RoboDK station: RBT23CS013(Yashashri_Kalekar).rdk

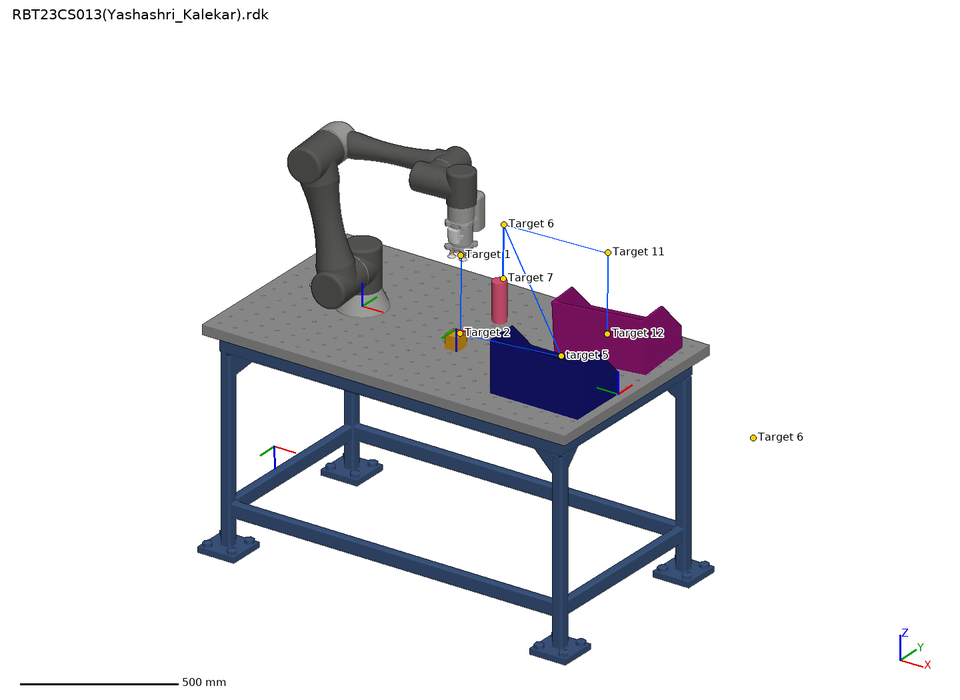
[picture v0: the station drawn from its stored meshes, robots at their saved joint values, targets as dots, program paths as lines]
Station RBT23CS013(Yashashri_Kalekar) (saved by RoboDK 5.9.2). Poses are relative to the parent item; angles as X-Y-Z fixed-axis rotations.
  - frame TM5-900 Base at (-216.63, 0, 0) mm
    - robot TM5-900: 6 axes, payload 4 kg, reach 900 mm, repeatability 0.1 mm, weight 30 kg
        modified DH rows (alpha deg, a mm, theta deg, d mm): 0, 0, 0, 145.2; 90, 0, 90, 0; 0, 429, 0, 0; 0, 411, -90, 122.3; -90, 0, 0, 106.5; 90, 0, 180, 114.15
        joint limits [-360, -180, -155, -180, -180, -270] to [360, 180, 155, 180, 180, 270]; home [0, 0, 90, -90, 90, 0]; saved at [4.776, -11.318, 99.736, 1.887, 89.639, -89.005]
      - tool SMC ZXP7A01-ZP25C-X1 Vacuum Gripper, TCP at (0, 0, 125) mm, size 88 x 106.8 x 127.9 mm
    - object Table 1400x800x800mm at (0, 0, 0) mm, size 1420 x 820 x 800 mm, geometry from Table.sld
  - frame Frame 2 at (811.01, -58.35, 0.44) mm, rotated rx 0 ry 0 rz 90.19 deg
    - object Bin Blue at (0, 0, 0) mm, size 225 x 337.5 x 191.2 mm, geometry from Bin-Blue.sld
  - frame Frame 3 at (181.66, -53.2, 51.85) mm, rotated rx -179.22 ry 0 rz 0 deg
    - object Cube 50mm at (-10, 0, 0) mm, size 50 x 50 x 50 mm, geometry from Cube.sld
    - target Target 1 (Cartesian target) at (42.39, 30.35, -286.08) mm, rotated rx 1.14 ry 0.35 rz 176.22 deg; joints [4.776, -11.318, 99.736, 1.887, 89.639, -89.005] of TM5-900
    - target Target 2 (Cartesian target) at (41.08, 35.92, -10.91) mm, rotated rx 1.14 ry 0.35 rz 176.22 deg; joints [4.546, 2.331, 129.082, -41.11, 89.638, -89.234] of TM5-900
    - target target 5 (Cartesian target) at (415.52, 10.86, -25.67) mm, rotated rx 1.14 ry 0.35 rz 176.22 deg; joints [4.198, 46.277, 61.378, -17.353, 89.636, -89.582] of TM5-900
    - object Bin Pink at (617.32, -365.19, 43.61) mm, rotated rx 177.31 ry 0 rz -94.05 deg, size 225 x 337.5 x 191.2 mm, geometry from Bin-Pink.sld
      - target Target 6 (Cartesian target) at (25.1, -231.08, -280.88) mm, rotated rx 1.14 ry 0.35 rz 176.22 deg; joints [37.917, -10.007, 98.873, 1.586, 89.865, -55.864] of TM5-900
      - target Target 6 (Cartesian target) at (25.1, -231.08, -280.88) mm, rotated rx 1.14 ry 0.35 rz 176.22 deg; joints [37.917, -10.007, 98.873, 1.586, 89.865, -55.864] of TM5-900
    - target Target 6 (Cartesian target) at (25.1, -231.08, -280.88) mm, rotated rx 1.14 ry 0.35 rz 176.22 deg; joints [37.917, -10.007, 98.873, 1.586, 89.865, -55.864] of TM5-900
    - target Target 7 (Cartesian target) at (24.19, -227.22, -89.78) mm, rotated rx 1.14 ry 0.35 rz 176.22 deg; joints [37.858, -4.045, 121.336, -26.84, 89.864, -55.923] of TM5-900
    - target Target 10 (Cartesian target) at (25.1, -231.08, -280.88) mm, rotated rx 1.14 ry 0.35 rz 176.22 deg; joints [37.917, -10.007, 98.873, 1.586, 89.865, -55.864] of TM5-900
    - target Target 11 (Cartesian target) at (408.79, -256.41, -278.53) mm, rotated rx 1.14 ry 0.35 rz 176.22 deg; joints [22.411, 53.381, 11.786, 25.233, 89.749, -71.369] of TM5-900
    - target Target 12 (Cartesian target) at (407.43, -250.65, 6.05) mm, rotated rx 1.14 ry 0.35 rz 176.22 deg; joints [22.324, 49.649, 59.362, -18.612, 89.748, -71.456] of TM5-900
    - frame Frame 4 at (0, 1000, 0) mm
      - object Cylinder 50x150mm at (18.29, -1213.2, -88.15) mm, size 50 x 50 x 150 mm, geometry from Cylinder-50x150mm.sld
  - program Prog1 (10 instructions, listed below)
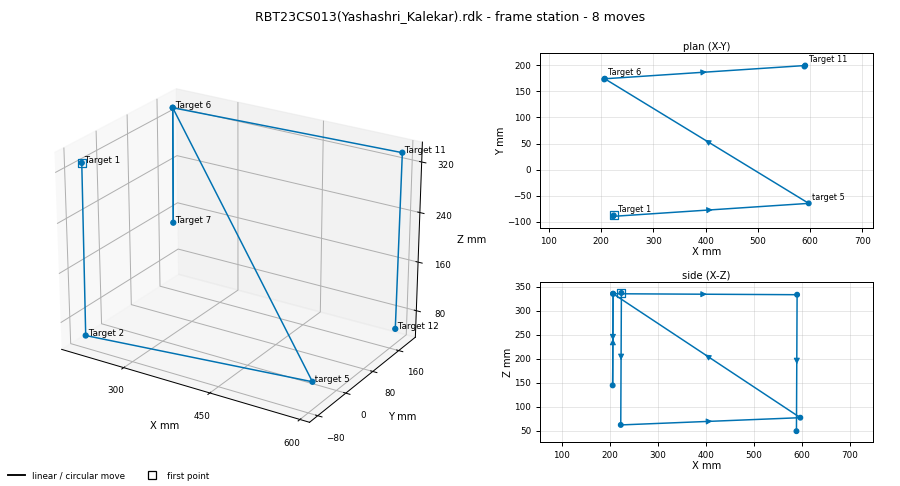
[picture p0: tool path of RBT23CS013(Yashashri_Kalekar).rdk in frame station, 8 of 8 moves have a stored position in this frame; points joined in program order, loops and branches not executed]

--- program Prog1 (robot TM5-900) ---
  Set Ref.: Frame 3
  Set Tool: SMC ZXP7A01-ZP25C-X1 Vacuum Gripper
  MoveJ (Target 1)
  MoveL (Target 2)
  MoveL (target 5)
  MoveL (Target 6)
  MoveL (Target 7)
  MoveL (Target 10)
  MoveL (Target 11)
  MoveL (Target 12)
